// TwinCAT 3 PLC project SuperBohrmachine
// ProgramVersion: 3.1.4023.0
// libraries:
//   Tc2_MC2, * (Beckhoff Automation GmbH)
//   Tc2_Standard, * (Beckhoff Automation GmbH)
//   Tc2_System, * (Beckhoff Automation GmbH)
//   Tc3_Module, * (Beckhoff Automation GmbH)
// project tree:
//   DUTs/ E_STATES_BOHRKOPF.TcDUT, E_STATES_SUPERBOHRMACHINE.TcDUT
//   / PlcTask.TcTTO, RecipeManager.TcRMO (not stored)
//   POUs/ AxesManager.TcPOU, Bohrkopf.TcPOU, I_SuperBohrmachine.TcIO, MAIN.TcPOU, SuperBohrmachine.TcCD (not stored), SuperBohrmachine.TcPOU
// (motion and I/O tree: see PLC project bohrmachine)
// real-time tasks:
//   TASK PlcTask: cycle T#10ms, priority 20, ADS port 350
//   TASK PlcTask1: cycle T#10ms, priority 21, ADS port 351
//   TASK PlcTask2: cycle T#10ms, priority 22, ADS port 352
//   TASK PlcTask3: cycle T#10ms, priority 23, ADS port 353
//   TASK ControllerTask: cycle T#10ms, priority 1, ADS port 354
//   TASK PlcTask4: cycle T#10ms, priority 24, ADS port 355
//   TASK PlcTask5: cycle T#10ms, priority 25, ADS port 356
// variable links:
//   SuperBohrmachine/SuperBohrmachine Instance <-> NC-Task 1 SAF/Axes/xAchse
//     PlcTask Inputs/MAIN.fbSuperBohrmachine.fbAxesManager.xAchse.NcToPlc <-> Outputs/ToPlc
//     PlcTask Outputs/MAIN.fbSuperBohrmachine.fbAxesManager.xAchse.PlcToNc <-> Inputs/FromPlc
//   SuperBohrmachine/SuperBohrmachine Instance <-> NC-Task 1 SAF/Axes/yAchse
//     PlcTask Inputs/MAIN.fbSuperBohrmachine.fbBohrkopf.axisRef.NcToPlc <-> Outputs/ToPlc
//     PlcTask Outputs/MAIN.fbSuperBohrmachine.fbBohrkopf.axisRef.PlcToNc <-> Inputs/FromPlc
//   SuperBohrmachine/SuperBohrmachine Instance <-> NC-Task 1 SAF/Axes/zAchse
//     PlcTask Inputs/MAIN.fbSuperBohrmachine.fbAxesManager.zAchse.NcToPlc <-> Outputs/ToPlc
//     PlcTask Outputs/MAIN.fbSuperBohrmachine.fbAxesManager.zAchse.PlcToNc <-> Inputs/FromPlc

CONFIGURATION SuperBohrmachine
    RESOURCE PLC ON TwinCAT3
        TASK PlcTask(INTERVAL := T#10ms, PRIORITY := 25);
        PROGRAM MAIN WITH PlcTask : MAIN;
    END_RESOURCE
END_CONFIGURATION

// ---- DUTs/E_STATES_BOHRKOPF.TcDUT
{attribute 'qualified_only'}
{attribute 'strict'}
TYPE E_STATES_BOHRKOPF :
(
	initializing := 0,
	stopped,
	stopping,
	ready,
	going_down,
	going_up
);
END_TYPE

// ---- DUTs/E_STATES_SUPERBOHRMACHINE.TcDUT
{attribute 'qualified_only'}
{attribute 'strict'}
TYPE E_STATES_SUPERBOHRMACHINE :
(
	initializing := 0,
	ready,
	moving,
	drilling,
	stopping,
	stopped,
	finishing
);
END_TYPE

// ---- POUs/I_SuperBohrmachine.TcIO
INTERFACE I_SuperBohrmachine

METHOD Bohren : HRESULT
END_METHOD

METHOD Start : HRESULT
VAR_INPUT
	config: REFERENCE TO ST_Config;
END_VAR
END_METHOD

METHOD Stop : HRESULT
VAR_INPUT
END_VAR
END_METHOD

END_INTERFACE

// ---- POUs/MAIN.TcPOU
PROGRAM MAIN
VAR
	fbSuperBohrmachine: SuperBohrmachine;
END_VAR

fbSuperBohrmachine();

END_PROGRAM

// ---- POUs/SuperBohrmachine.TcPOU
FUNCTION_BLOCK SuperBohrmachine IMPLEMENTS I_SuperBohrmachine
VAR_INPUT
END_VAR
VAR_OUTPUT
END_VAR
VAR
	fbBohrkopf: Bohrkopf;
	fbAxesManager: AxesManager;
	stConfig: ST_Config;
	
	eZustand: E_STATES_SUPERBOHRMACHINE := E_STATES_SUPERBOHRMACHINE.stopped;
	
	// Stop-Command set via outside call?
	bDoStop: BOOL := FALSE;
	
	// anzufahrende Punkte
	aPunkte: ARRAY [0..3] OF ST_2DPoint;
	nCurIdx: USINT := 0;
END_VAR

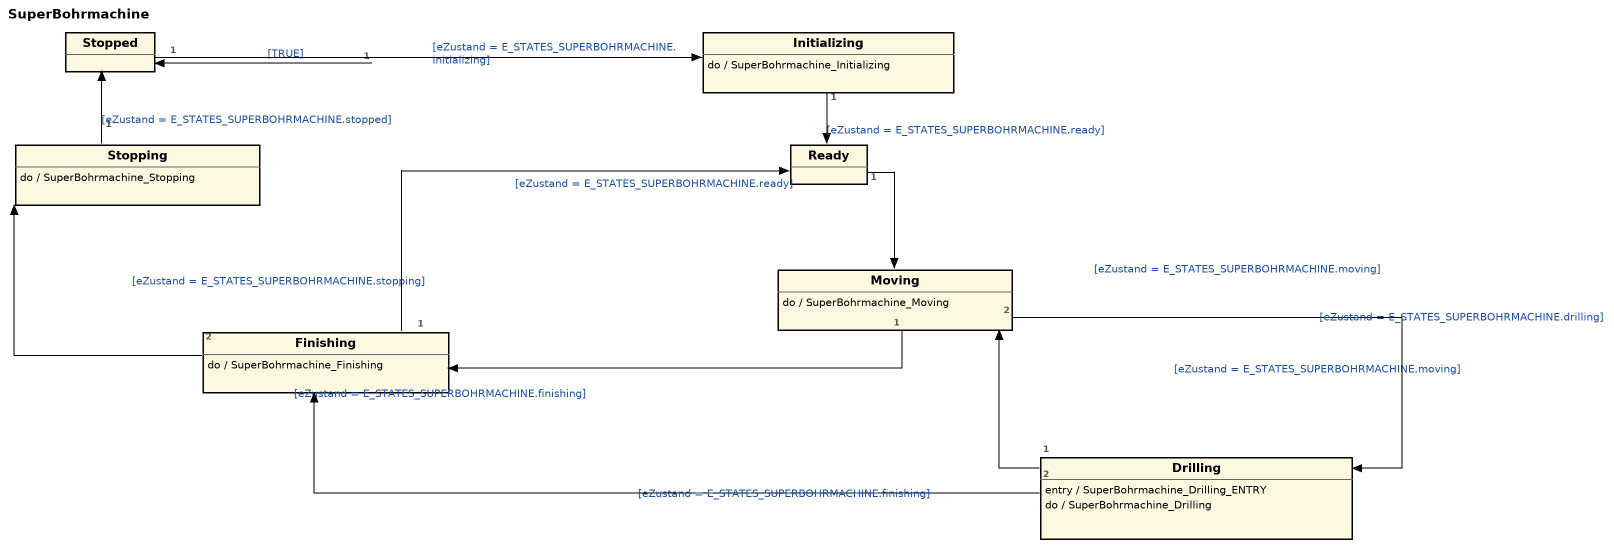
STATECHART SuperBohrmachine  // abortable
    START StartState1
    STATE Stopped
    STATE Initializing
        do / SuperBohrmachine_Initializing
    STATE Stopping
        do / SuperBohrmachine_Stopping
    STATE Ready
    STATE Moving
        do / SuperBohrmachine_Moving
    STATE Finishing
        do / SuperBohrmachine_Finishing
    STATE Drilling
        entry / SuperBohrmachine_Drilling_ENTRY
        do / SuperBohrmachine_Drilling
    StartState1 -> Stopped [TRUE] // priority 1, on completion
    Stopped -> Initializing [eZustand = E_STATES_SUPERBOHRMACHINE.initializing] // priority 1
    Initializing -> Ready [eZustand = E_STATES_SUPERBOHRMACHINE.ready] // priority 1
    Stopping -> Stopped [eZustand = E_STATES_SUPERBOHRMACHINE.stopped] // priority 1
    Ready -> Moving [eZustand = E_STATES_SUPERBOHRMACHINE.moving] // priority 1
    Moving -> Finishing [eZustand = E_STATES_SUPERBOHRMACHINE.finishing] // priority 1
    Moving -> Drilling [eZustand = E_STATES_SUPERBOHRMACHINE.drilling] // priority 2
    Finishing -> Ready [eZustand = E_STATES_SUPERBOHRMACHINE.ready] // priority 1
    Finishing -> Stopping [eZustand = E_STATES_SUPERBOHRMACHINE.stopping] // priority 2
    Drilling -> Moving [eZustand = E_STATES_SUPERBOHRMACHINE.moving] // priority 1
    Drilling -> Finishing [eZustand = E_STATES_SUPERBOHRMACHINE.finishing] // priority 2
END_STATECHART

METHOD Bohren : HRESULT
CASE eZustand OF
	E_STATES_SUPERBOHRMACHINE.ready:
		THIS^.eZustand := E_STATES_SUPERBOHRMACHINE.moving;
		Bohren := S_OK;
		
	ELSE
		Bohren := S_FALSE;

END_CASE
END_METHOD

PROPERTY PUBLIC Config : ST_Config
SET
VAR
	rBreite: LREAL;
	rLaenge: LREAL;
	rAbstand: LREAL := 10;
END_VAR
stConfig := Config;

// Punkte berechnen
rBreite := stConfig.rBreite;
rLaenge := stConfig.rLaenge;

// Punkt 1
aPunkte[0].x := rAbstand;
aPunkte[0].y := rAbstand;

// Punkt 2
aPunkte[1].x := 10;
aPunkte[1].y := rBreite - rAbstand;

// Punkt 3
aPunkte[2].x := rLaenge - rAbstand;
aPunkte[2].y := rBreite - rAbstand;

// Punkt 4
aPunkte[3].x := rLaenge - rAbstand;
aPunkte[3].y := rAbstand;

fbBohrkopf.Config REF= stConfig;
END_SET
END_PROPERTY

METHOD Start : HRESULT
VAR_INPUT
	config: REFERENCE TO ST_Config;
END_VAR
CASE eZustand OF
	E_STATES_SUPERBOHRMACHINE.stopped:
		// Konfiguration setzen
		THIS^.Config := config;
		// Anlage starten
		THIS^.eZustand := E_STATES_SUPERBOHRMACHINE.initializing;
		Start := S_PENDING;
		
	E_STATES_SUPERBOHRMACHINE.ready:
		Start := S_OK;
		
	ELSE
		Start := S_PENDING;
	
END_CASE
END_METHOD

METHOD Stop : HRESULT
CASE eZustand OF
	// Anlage gestoppt
	E_STATES_SUPERBOHRMACHINE.stopped:
		Stop := S_OK;
	
	E_STATES_SUPERBOHRMACHINE.finishing:
		// Stop während normalem Finishing
		THIS^.bDoStop := TRUE;
		Stop := S_PENDING;

	E_STATES_SUPERBOHRMACHINE.stopping:
		Stop := S_PENDING;

	ELSE
		// Anlage stoppen
		THIS^.bDoStop := TRUE;
		THIS^.eZustand := E_STATES_SUPERBOHRMACHINE.finishing;
		
END_CASE
END_METHOD

METHOD PRIVATE SuperBohrmachine_Drilling : BOOL
VAR_INPUT
END_VAR

IF fbBohrkopf.Ready THEN
	// fertig gebohrt
	eZustand := E_STATES_SUPERBOHRMACHINE.moving;
END_IF
END_METHOD

METHOD PRIVATE SuperBohrmachine_Drilling_ENTRY : BOOL
VAR_INPUT
END_VAR
fbBohrkopf.Bohren();
END_METHOD

METHOD PRIVATE SuperBohrmachine_Finishing : BOOL
VAR
	stHomePoint: ST_2DPoint := (x := 0, y := 0);
END_VAR
VAR_INST
	bAxesHomeDone: BOOL := FALSE;
	bBohrkopfUpDone: BOOL := FALSE;
END_VAR
(*
1. Bohrkopf hochfahren
2. AxesManager zum Nullpunkt fahren
3. bDoStop = TRUE ? 'stopping' : 'ready'
*)

fbBohrkopf.GoUp(Done => bBohrkopfUpDone);

IF bBohrkopfUpDone THEN
	fbAxesManager.GoTo(stHomePoint, Done => bAxesHomeDone);
	IF bAxesHomeDone THEN
		bAxesHomeDone := FALSE;
		bBohrkopfUpDone := FALSE;
		// Anlage stoppen oder Bearbeitung fertig?
		IF bDoStop THEN
			eZustand := E_STATES_SUPERBOHRMACHINE.stopping;
		ELSE
			eZustand := E_STATES_SUPERBOHRMACHINE.ready;
		END_IF
	END_IF
END_IF
END_METHOD

METHOD PRIVATE SuperBohrmachine_Initializing : BOOL
VAR_INPUT
END_VAR
(*
- AxesManager initialisieren
- Bohrkopf initialisieren
*)

fbAxesManager.Init();
fbBohrkopf.Init();

IF fbAxesManager.Initialized AND fbBohrkopf.Initialized THEN
	// Anlage initialisiert
	eZustand := E_STATES_SUPERBOHRMACHINE.ready;
END_IF
END_METHOD

METHOD PRIVATE SuperBohrmachine_Moving : BOOL
VAR_INPUT
END_VAR
IF nCurIdx = 4 THEN
	// letzter Punkt wurde gebohrt => State 'finishing'
	nCurIdx := 0;
	eZustand := E_STATES_SUPERBOHRMACHINE.finishing;
ELSE
	// Zum Punkt fahren => State 'drilling'
	IF fbAxesManager.GoTo(aPunkte[nCurIdx]) THEN
		nCurIdx := nCurIdx + 1;
		eZustand := E_STATES_SUPERBOHRMACHINE.drilling;
	END_IF
END_IF
END_METHOD

METHOD PRIVATE SuperBohrmachine_Stopping : BOOL
VAR CONSTANT
	stHomePoint: ST_2DPoint := (x := 0, y := 0);
END_VAR
VAR_INST
	bAxesStopDone: BOOL := FALSE;
	bBohrkopfStopDone: BOOL := FALSE;
END_VAR
(*
- Bohrkopf-Achsen stoppen
- AxesManager stop
*)

fbBohrkopf.Stop();
fbAxesManager.Stop();


IF fbAxesManager.Stopped AND fbBohrkopf.Stopped THEN
	bDoStop := FALSE;
	eZustand := E_STATES_SUPERBOHRMACHINE.stopped;
END_IF
END_METHOD

END_FUNCTION_BLOCK

// ---- POUs/Bohrkopf.TcPOU
FUNCTION_BLOCK Bohrkopf
VAR_INPUT
END_VAR
VAR_OUTPUT
	Done: BOOL := FALSE;
	Stopped: BOOL := TRUE;
	Initialized: BOOL := FALSE;
END_VAR
VAR
	axisRef: AXIS_REF;
	fbMcMove: MC_MoveAbsolute;
	fbMcPower: MC_Power;
	fbMcStop: MC_Stop;
	eZustand: E_STATES_BOHRKOPF := E_STATES_BOHRKOPF.stopped;
	
	stConfig: REFERENCE TO ST_Config;
	
	// Stop-Command set via outside call?
	bDoStop: BOOL := FALSE;
END_VAR

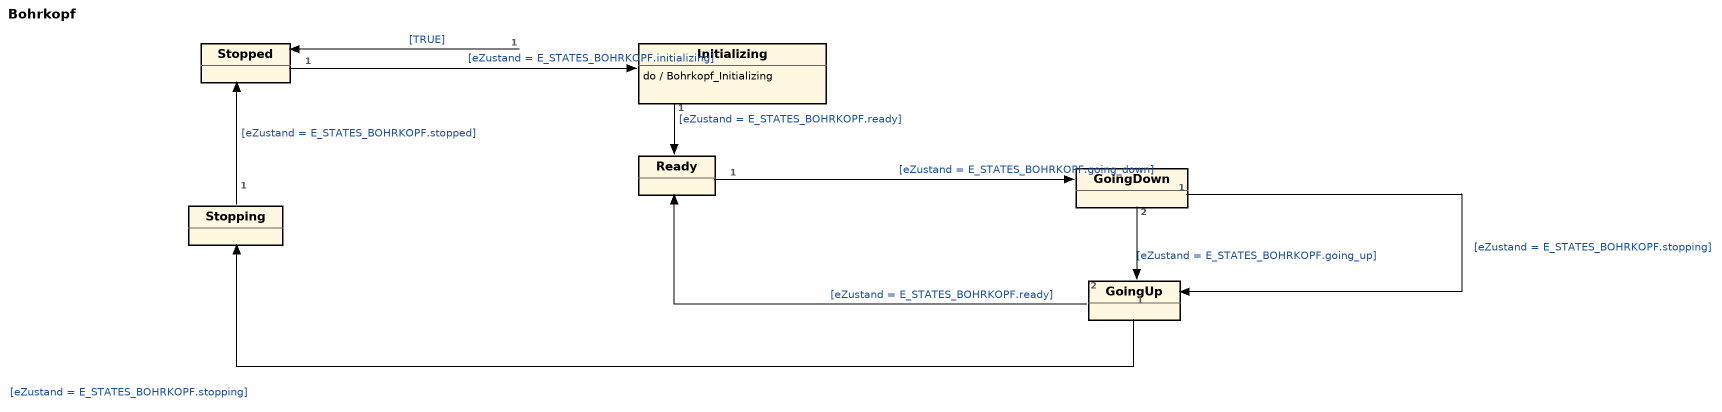
STATECHART Bohrkopf  // abortable
    START StartState1
    STATE Stopped
    STATE Initializing
        do / Bohrkopf_Initializing
    STATE Ready
    STATE GoingDown
    STATE Stopping
    STATE GoingUp
    StartState1 -> Stopped [TRUE] // priority 1, on completion
    Stopped -> Initializing [eZustand = E_STATES_BOHRKOPF.initializing] // priority 1
    Initializing -> Ready [eZustand = E_STATES_BOHRKOPF.ready] // priority 1
    Ready -> GoingDown [eZustand = E_STATES_BOHRKOPF.going_down] // priority 1
    GoingDown -> GoingUp [eZustand = E_STATES_BOHRKOPF.stopping] // priority 1
    GoingDown -> GoingUp [eZustand = E_STATES_BOHRKOPF.going_up] // priority 2
    Stopping -> Stopped [eZustand = E_STATES_BOHRKOPF.stopped] // priority 1
    GoingUp -> Stopping [eZustand = E_STATES_BOHRKOPF.stopping] // priority 1
    GoingUp -> Ready [eZustand = E_STATES_BOHRKOPF.ready] // priority 2
END_STATECHART

METHOD PUBLIC Bohren : HRESULT
VAR_INPUT
END_VAR
CASE eZustand OF
	E_STATES_BOHRKOPF.ready:
		// bohren starten
		eZustand := E_STATES_BOHRKOPF.going_down;
		Bohren := S_PENDING;
		
	ELSE
		// bohrend
		Bohren := S_PENDING;
END_CASE
END_METHOD

METHOD Bohrkopf_Initializing : HRESULT
VAR_INPUT
END_VAR
axisRef.ReadStatus();

fbMcPower(
	Axis := axisRef,
	Enable := TRUE,
	Enable_Positive := TRUE,
	Enable_Negative := TRUE
);

IF fbMcPower.Status THEN
	THIS^.Initialized := TRUE;
	THIS^.eZustand := E_STATES_BOHRKOPF.ready;
END_IF
END_METHOD

PROPERTY PUBLIC Config : REFERENCE TO ST_Config
SET
THIS^.stConfig := Config;
END_SET
END_PROPERTY

METHOD PUBLIC GoUp : BOOL
VAR_INPUT
END_VAR
VAR_OUTPUT
	Done: BOOL := FALSE;
END_VAR
// Bohrkopf in Ausgangsposition hochfahren
END_METHOD

PROPERTY PUBLIC Ready : BOOL
GET
Ready := THIS^.eZustand = E_STATES_BOHRKOPF.ready;
END_GET
END_PROPERTY

METHOD PUBLIC Stop : BOOL
VAR_INPUT
END_VAR
//CASE eZustand OF
//	E_STATES_BOHRKOPF.ready:
//		Stop := TRUE;
		
//	ELSE
//		Stop := FALSE;
//END_CASE
END_METHOD

END_FUNCTION_BLOCK

// ---- POUs/AxesManager.TcPOU
FUNCTION_BLOCK AxesManager
VAR_INPUT
END_VAR
VAR
	xAchse: AXIS_REF;
	zAchse: AXIS_REF;
	fbMcPowerX: MC_Power;
	fbMcPowerZ: MC_Power;
	fbMcMoveX: MC_MoveAbsolute;
	fbMcMoveZ: MC_MoveAbsolute;
END_VAR

xAchse.ReadStatus();
zAchse.ReadStatus();

METHOD PUBLIC GoTo : BOOL
VAR_INPUT
	stCurPoint: REFERENCE TO ST_2DPoint;
END_VAR
VAR_OUTPUT
	Done: BOOL := FALSE;
END_VAR
fbMcMoveX(
	Axis := xAchse,
	Execute := TRUE,
	Position := stCurPoint.x
);

fbMcMoveZ(
	Axis := zAchse,
	Execute := TRUE,
	Position := stCurPoint.y
);

// Punkt angefahren
Done := fbMcMoveX.Done AND fbMcMoveZ.Done; 

IF Done THEN
	// Bausteine einmal falsen
	fbMcMoveX(Axis := xAchse, Execute := FALSE);
	fbMcMoveZ(Axis := zAchse, Execute := FALSE);
END_IF
END_METHOD

METHOD PUBLIC Init : BOOL
VAR_INPUT
END_VAR
fbMcPowerX(
	Axis := xAchse,
	Enable := TRUE,
	Enable_Positive := TRUE,
	Enable_Negative := TRUE
);

fbMcPowerZ(
	Axis := zAchse,
	Enable := TRUE,
	Enable_Positive := TRUE,
	Enable_Negative := TRUE
);

fbMcPowerX.Status;
END_METHOD

PROPERTY PUBLIC Initialized : BOOL
GET
// Beide Achsen bereit? => TRUE
Initialized := fbMcPowerX.Status AND fbMcPowerZ.Status;
END_GET
END_PROPERTY

METHOD PUBLIC Stop : BOOL
VAR_INPUT
END_VAR
fbMcPowerX(
	Axis := xAchse,
	Enable := FALSE
);

fbMcPowerZ(
	Axis := zAchse,
	Enable := FALSE
);
END_METHOD

PROPERTY PUBLIC Stopped : BOOL
GET
// Beide Achsen gestoppt? => TRUE
Stopped := NOT fbMcPowerX.Status AND NOT fbMcPowerZ.Status;
END_GET
END_PROPERTY

END_FUNCTION_BLOCK
